(* Schneider Machine Expert - Basic project exercise_3.4, file version 2.9.0.0 *)
(* ProjectInformations: Name=Novo projeto *)

HARDWARE
  Cpu 0: TM221M16R/G
  ModuleExtensionObject 0: TM3DM24R/G
  EthernetConfiguration: NetworkName=M221, IpAllocationMode=FixedAddress, IpAddress=0.0.0.0, SubnetMask=0.0.0.0
  SerialLineConfiguration: Baud=Baud19200, Parity=ParityEven, DataBits=DataBits8, StopBits=StopBits1, PhysicalMedium=PhysicalMediumRs485, TransmissionMode=TransmissionModeModbusRtu, SlaveId=1, Addressing=SlaveAddressing
  MastTask: UsePeriodScanMode=false, PeriodScan=100
  FastTask: Period=255
  CpuBehavior: StartingMode=StartAsPreviousState, AutoSaveRamOnEeprom=true, WatchdogPeriod=250

SYMBOLS  (address, symbol, comment, settings)
  %M0       SIG_IN_L_ATU
  %M1       SIG_IN_L_DESA
  %M2       SIG_IN_D_ATU
  %M3       SIG_IN_D_DESA
  %M4       SIG_IN_SEN_A
  %M5       SIG_IN_SEN_B
  %M6       SIG_IN_SEN_C
  %M7       SIG_IN_SEL_P
  %M8       SIG_IN_SEL_M
  %M9       SIG_IN_SEL_G
  %M15      SIG_SEN_ERR
  %M20      SIG_ATU_E_LIGA
  %M21      SIG_ATU_E_DESL
  %M22      SIG_ALA_AL_LIGA
  %M23      SIG_ALA_AL_DESL
  %I0.0     IN_L_ATU
  %I0.1     IN_L_DESA
  %I0.2     IN_D_ATU
  %I0.3     IN_D_DESA
  %I0.5     IN_SEN_A
  %I0.6     IN_SEN_B
  %I0.7     IN_SEN_C
  %Q0.1     OUT_ATU_E
  %Q0.2     OUT_ALA_AL
  %I1.0     IN_SEL_P
  %I1.1     IN_SEL_M
  %I1.2     IN_SEL_G

POU Entradas
  (* SectionNumber=1 *)

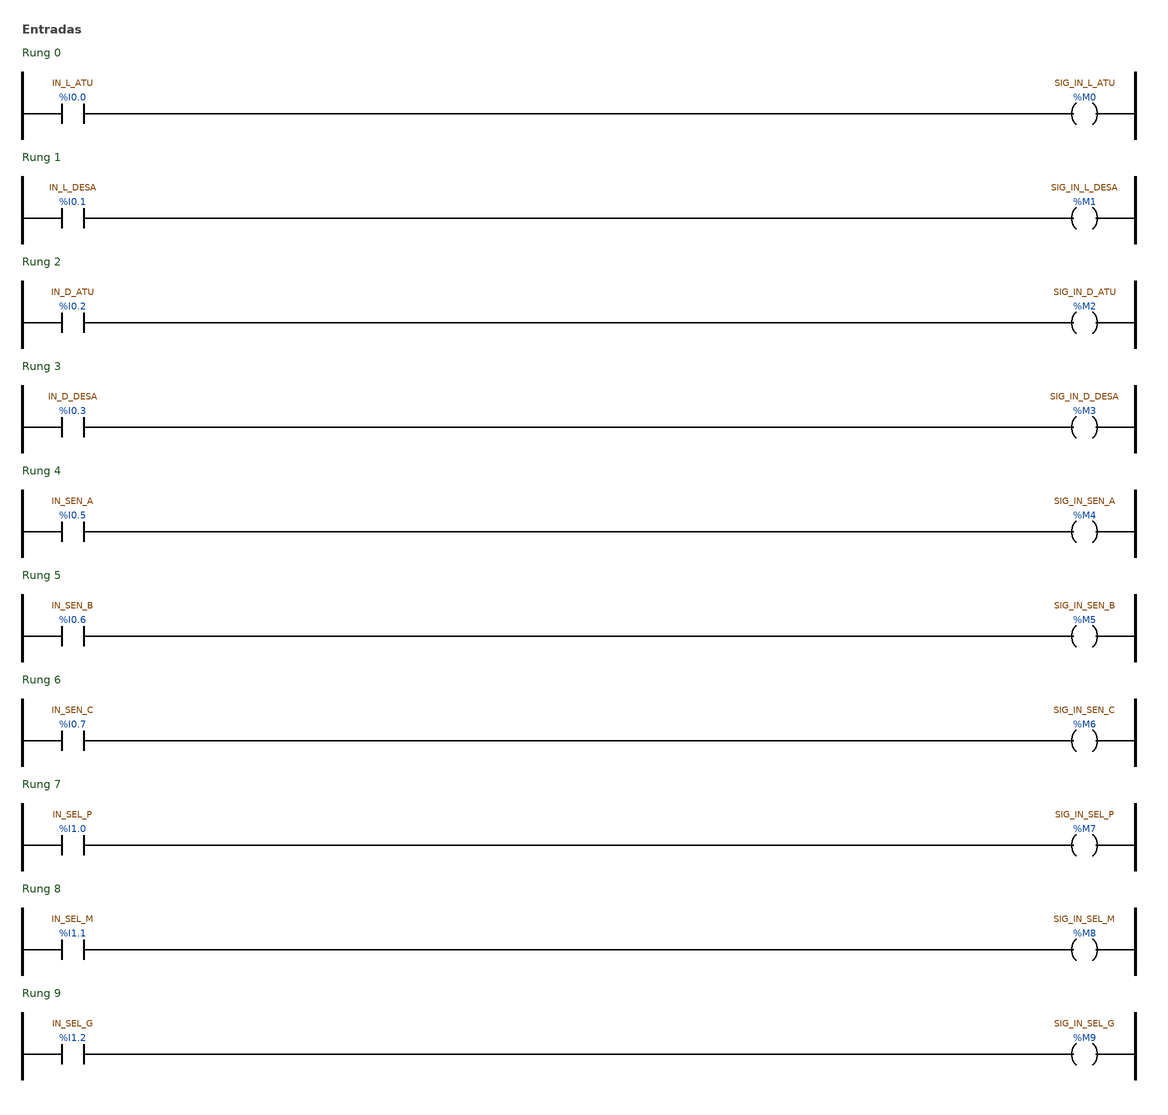

// Rung 0
  LD %I0.0                (* IN_L_ATU *)
  ST %M0                  (* SIG_IN_L_ATU *)
  // as ST:
  //   SIG_IN_L_ATU := IN_L_ATU;

// Rung 1
  LD %I0.1                (* IN_L_DESA *)
  ST %M1                  (* SIG_IN_L_DESA *)
  // as ST:
  //   SIG_IN_L_DESA := IN_L_DESA;

// Rung 2
  LD %I0.2                (* IN_D_ATU *)
  ST %M2                  (* SIG_IN_D_ATU *)
  // as ST:
  //   SIG_IN_D_ATU := IN_D_ATU;

// Rung 3
  LD %I0.3                (* IN_D_DESA *)
  ST %M3                  (* SIG_IN_D_DESA *)
  // as ST:
  //   SIG_IN_D_DESA := IN_D_DESA;

// Rung 4
  LD %I0.5                (* IN_SEN_A *)
  ST %M4                  (* SIG_IN_SEN_A *)
  // as ST:
  //   SIG_IN_SEN_A := IN_SEN_A;

// Rung 5
  LD %I0.6                (* IN_SEN_B *)
  ST %M5                  (* SIG_IN_SEN_B *)
  // as ST:
  //   SIG_IN_SEN_B := IN_SEN_B;

// Rung 6
  LD %I0.7                (* IN_SEN_C *)
  ST %M6                  (* SIG_IN_SEN_C *)
  // as ST:
  //   SIG_IN_SEN_C := IN_SEN_C;

// Rung 7
  LD %I1.0                (* IN_SEL_P *)
  ST %M7                  (* SIG_IN_SEL_P *)
  // as ST:
  //   SIG_IN_SEL_P := IN_SEL_P;

// Rung 8
  LD %I1.1                (* IN_SEL_M *)
  ST %M8                  (* SIG_IN_SEL_M *)
  // as ST:
  //   SIG_IN_SEL_M := IN_SEL_M;

// Rung 9
  LD %I1.2                (* IN_SEL_G *)
  ST %M9                  (* SIG_IN_SEL_G *)
  // as ST:
  //   SIG_IN_SEL_G := IN_SEL_G;

POU Lógicas
  (* SectionNumber=2 *)

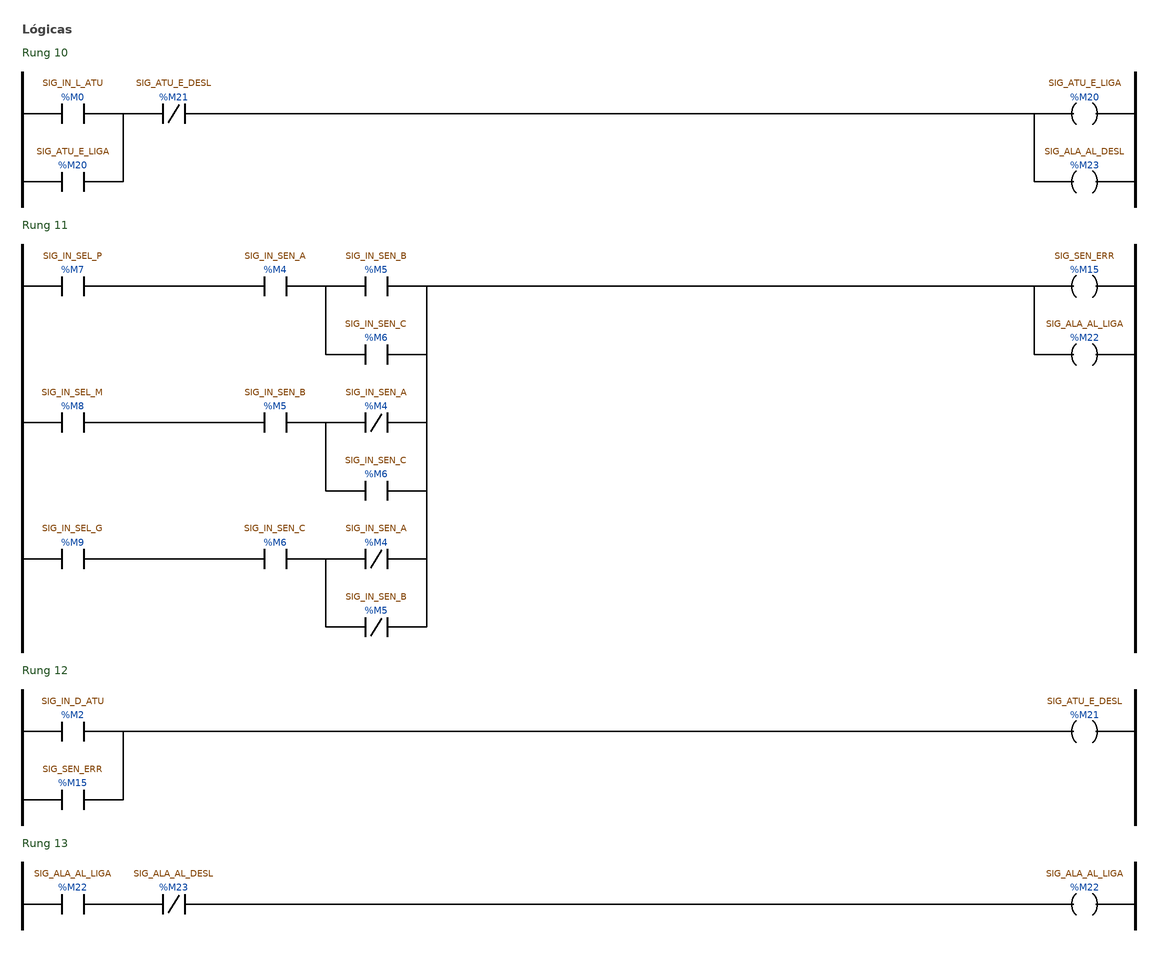

// Rung 10
  LD %M0                  (* SIG_IN_L_ATU *)
  OR %M20                 (* SIG_ATU_E_LIGA *)
  ANDN %M21               (* SIG_ATU_E_DESL *)
  ST %M20                 (* SIG_ATU_E_LIGA *)
  ST %M23                 (* SIG_ALA_AL_DESL *)
  // as ST:
  //   _t1 := (SIG_IN_L_ATU OR SIG_ATU_E_LIGA) AND NOT SIG_ATU_E_DESL;
  //   SIG_ATU_E_LIGA := _t1;
  //   SIG_ALA_AL_DESL := _t1;

// Rung 11
  LD %M7                  (* SIG_IN_SEL_P *)
  AND %M4                 (* SIG_IN_SEN_A *)
  AND( %M5                (* SIG_IN_SEN_B *)
  OR %M6                  (* SIG_IN_SEN_C *)
  )
  OR( %M8                 (* SIG_IN_SEL_M *)
  AND %M5                 (* SIG_IN_SEN_B *)
  AND(N %M4               (* SIG_IN_SEN_A *)
  OR %M6                  (* SIG_IN_SEN_C *)
  )
  )
  OR( %M9                 (* SIG_IN_SEL_G *)
  AND %M6                 (* SIG_IN_SEN_C *)
  AND(N %M4               (* SIG_IN_SEN_A *)
  ORN %M5                 (* SIG_IN_SEN_B *)
  )
  )
  ST %M15                 (* SIG_SEN_ERR *)
  ST %M22                 (* SIG_ALA_AL_LIGA *)
  // as ST:
  //   SIG_SEN_ERR := SIG_IN_SEL_P AND SIG_IN_SEN_A AND (SIG_IN_SEN_B OR SIG_IN_SEN_C) OR SIG_IN_SEL_M AND SIG_IN_SEN_B AND (NOT SIG_IN_SEN_A OR SIG_IN_SEN_C) OR SIG_IN_SEL_G AND SIG_IN_SEN_C AND (NOT SIG_IN_SEN_A OR NOT SIG_IN_SEN_B);
  //   SIG_ALA_AL_LIGA := SIG_IN_SEL_P AND SIG_IN_SEN_A AND (SIG_IN_SEN_B OR SIG_IN_SEN_C) OR SIG_IN_SEL_M AND SIG_IN_SEN_B AND (NOT SIG_IN_SEN_A OR SIG_IN_SEN_C) OR SIG_IN_SEL_G AND SIG_IN_SEN_C AND (NOT SIG_IN_SEN_A OR NOT SIG_IN_SEN_B);

// Rung 12
  LD %M2                  (* SIG_IN_D_ATU *)
  OR %M15                 (* SIG_SEN_ERR *)
  ST %M21                 (* SIG_ATU_E_DESL *)
  // as ST:
  //   SIG_ATU_E_DESL := SIG_IN_D_ATU OR SIG_SEN_ERR;

// Rung 13
  LD %M22                 (* SIG_ALA_AL_LIGA *)
  ANDN %M23               (* SIG_ALA_AL_DESL *)
  ST %M22                 (* SIG_ALA_AL_LIGA *)
  // as ST:
  //   SIG_ALA_AL_LIGA := SIG_ALA_AL_LIGA AND NOT SIG_ALA_AL_DESL;

POU Saídas
  (* SectionNumber=3 *)

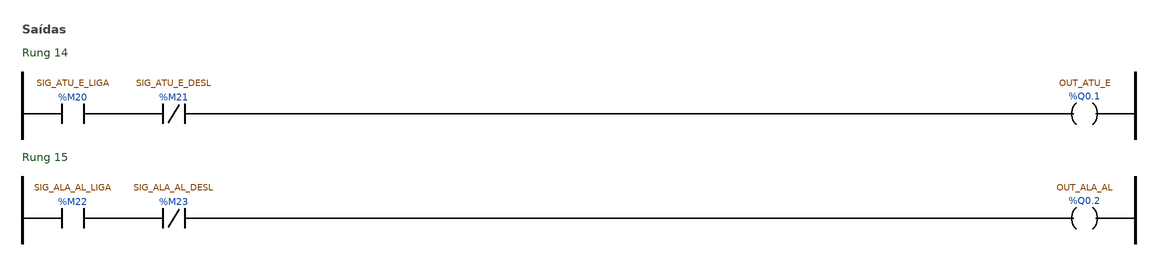

// Rung 14
  LD %M20                 (* SIG_ATU_E_LIGA *)
  ANDN %M21               (* SIG_ATU_E_DESL *)
  ST %Q0.1                (* OUT_ATU_E *)
  // as ST:
  //   OUT_ATU_E := SIG_ATU_E_LIGA AND NOT SIG_ATU_E_DESL;

// Rung 15
  LD %M22                 (* SIG_ALA_AL_LIGA *)
  ANDN %M23               (* SIG_ALA_AL_DESL *)
  ST %Q0.2                (* OUT_ALA_AL *)
  // as ST:
  //   OUT_ALA_AL := SIG_ALA_AL_LIGA AND NOT SIG_ALA_AL_DESL;
